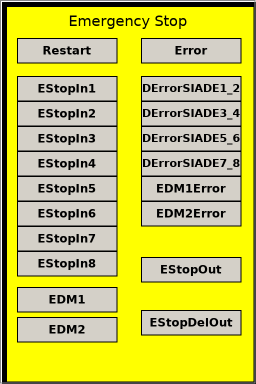
VISUALIZATION V_PH_ESTOP  // 256x384
VAR_INPUT
	stSafetyEStop				: ST_SAFETY_FBESTOP;
END_VAR
    Rectangle (2,2 256x384), colour toggle: stSafetyEStop.bGeneralError
    Label (53,6 150x30), "Emergency Stop"
    RoundedRectangle (17,38 100x25), "Restart", colour toggle: stSafetyEStop.uStatus.stStatusWords.wInputs.0
    RoundedRectangle (17,126 100x25), "EStopIn3", colour toggle: stSafetyEStop.uStatus.stStatusWords.wInputs.10
    RoundedRectangle (17,151 100x25), "EStopIn4", colour toggle: stSafetyEStop.uStatus.stStatusWords.wInputs.11
    RoundedRectangle (17,176 100x25), "EStopIn5", colour toggle: stSafetyEStop.uStatus.stStatusWords.wInputs.12
    RoundedRectangle (17,201 100x25), "EStopIn6", colour toggle: stSafetyEStop.uStatus.stStatusWords.wInputs.13
    RoundedRectangle (17,226 100x25), "EStopIn7", colour toggle: stSafetyEStop.uStatus.stStatusWords.wInputs.14
    RoundedRectangle (17,251 100x25), "EStopIn8", colour toggle: stSafetyEStop.uStatus.stStatusWords.wInputs.15
    RoundedRectangle (17,101 100x25), "EStopIn2", colour toggle: stSafetyEStop.uStatus.stStatusWords.wInputs.9
    RoundedRectangle (17,76 100x25), "EStopIn1", colour toggle: stSafetyEStop.uStatus.stStatusWords.wInputs.8
    RoundedRectangle (141,76 100x25), "DiscError1_2", colour toggle: stSafetyEStop.uStatus.stStatusWords.wDiagnosis.0, invisible if: NOT stSafetyEStop.uStatus.stStatusWords.wDiagnosis.0
    RoundedRectangle (141,101 100x25), "DicsError3_4", colour toggle: stSafetyEStop.uStatus.stStatusWords.wDiagnosis.1, invisible if: NOT stSafetyEStop.uStatus.stStatusWords.wDiagnosis.1
    RoundedRectangle (141,126 100x25), "DiscError5_6", colour toggle: stSafetyEStop.uStatus.stStatusWords.wDiagnosis.2, invisible if: NOT stSafetyEStop.uStatus.stStatusWords.wDiagnosis.2
    RoundedRectangle (141,176 100x25), "EDM1Error", colour toggle: stSafetyEStop.uStatus.stStatusWords.wDiagnosis.4, invisible if: NOT stSafetyEStop.uStatus.stStatusWords.wDiagnosis.4
    RoundedRectangle (141,310 100x25), "EStopDelOut", colour toggle: stSafetyEStop.uStatus.stStatusWords.wOutputs.2
    RoundedRectangle (141,38 100x25), "Error", colour toggle: stSafetyEStop.uStatus.stStatusWords.wOutputs.0
    RoundedRectangle (141,151 100x25), "DiscError7_8", colour toggle: stSafetyEStop.uStatus.stStatusWords.wDiagnosis.3, invisible if: NOT stSafetyEStop.uStatus.stStatusWords.wDiagnosis.3
    RoundedRectangle (141,257 100x25), "EStopOut", colour toggle: stSafetyEStop.uStatus.stStatusWords.wOutputs.1
    RoundedRectangle (17,287 100x25), "EDM1", colour toggle: stSafetyEStop.uStatus.stStatusWords.wInputs.1
    RoundedRectangle (17,317 100x25), "EDM2", colour toggle: stSafetyEStop.uStatus.stStatusWords.wInputs.2
    RoundedRectangle (141,76 100x25), "DErrorSIADE1_2", colour toggle: stSafetyEStop.uStatus.stStatusWords.wDiagnosis.8, invisible if: NOT stSafetyEStop.uStatus.stStatusWords.wDiagnosis.8
    RoundedRectangle (141,101 100x25), "DErrorSIADE3_4", colour toggle: stSafetyEStop.uStatus.stStatusWords.wDiagnosis.9, invisible if: NOT stSafetyEStop.uStatus.stStatusWords.wDiagnosis.9
    RoundedRectangle (141,126 100x25), "DErrorSIADE5_6", colour toggle: stSafetyEStop.uStatus.stStatusWords.wDiagnosis.10, invisible if: NOT stSafetyEStop.uStatus.stStatusWords.wDiagnosis.10
    RoundedRectangle (141,151 100x25), "DErrorSIADE7_8", colour toggle: stSafetyEStop.uStatus.stStatusWords.wDiagnosis.11, invisible if: NOT stSafetyEStop.uStatus.stStatusWords.wDiagnosis.11
    RoundedRectangle (141,201 100x25), "EDM2Error", colour toggle: stSafetyEStop.uStatus.stStatusWords.wDiagnosis.5, invisible if: NOT stSafetyEStop.uStatus.stStatusWords.wDiagnosis.5
    Textfield (17,354 234x25), text list: 'TL_FbState', text index: stSafetyEStop.eState
END_VISUALIZATION

(* stored: Version 1.1.0.1, ProductVersion 3.1.4024.4
   Visu V_PH_ESTOP: Id {3284071d-1f8d-4d2e-9ef5-6d581d763251} *)
